// TIA Portal V18 export
FUNCTION "Motor_control_FC" : Void   // FC1, LAD
{ S7_Optimized_Access := 'TRUE' }
VERSION : 0.1
// stored: AutoNumber true, IsIECCheckEnabled false, SetENOAutomatically false, UDAEnableTagReadback false
BEGIN

REGION Network 1
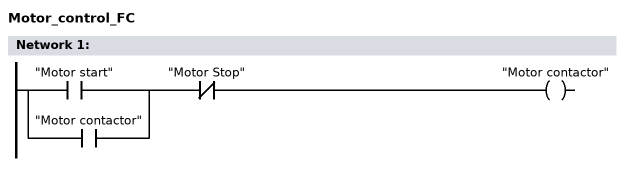
   RUNG wire#powerrail
      Contact( "Motor start" )
      wire#w1
      I_Contact( "Motor Stop" )
      Coil( "Motor contactor" )
   END_RUNG
   RUNG wire#powerrail
      Contact( "Motor contactor" )
   END_RUNG wire#w1
   // the same network as SCL:
   "Motor contactor" := ("Motor start" OR "Motor contactor") AND NOT "Motor Stop";
END_REGION
END_FUNCTION
